FUNCTION_BLOCK SECOND_ORDER_SYSTEM_SS (* 2nd ordem system y'' + K2y' + K1y = K*Xin *)
  (* Standard: 61499-2 *)
  (* Version 11-01-12, GASR *)
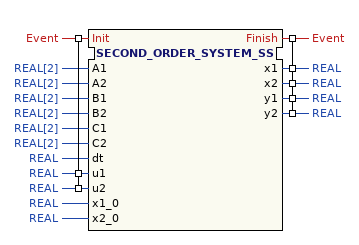
  EVENT_INPUT
    Init WITH u1, u2;
  END_EVENT
  EVENT_OUTPUT
    Finish WITH x1, x2, y1, y2;
  END_EVENT
  VAR_INPUT
    A1 : ARRAY [0..1] OF REAL; (* First row of matrix A *)
    A2 : ARRAY [0..1] OF REAL; (* Second row of matrix A *)
    B1 : ARRAY [0..1] OF REAL; (* First row of matrix B *)
    B2 : ARRAY [0..1] OF REAL; (* Second row of matrix B *)
    C1 : ARRAY [0..1] OF REAL; (* First row of matrix C *)
    C2 : ARRAY [0..1] OF REAL; (* Second row of matrix C *)
    dt : REAL;
    u1 : REAL;
    u2 : REAL;
    x1_0 : REAL; (* condicao inicial *)
    x2_0 : REAL;
  END_VAR
  VAR_OUTPUT
    x1 : REAL;
    x2 : REAL;
    y1 : REAL;
    y2 : REAL;
  END_VAR
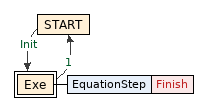
  EC_STATES
    Exe : EquationStep -> Finish;
    START;
  END_STATES
  EC_TRANSITIONS
    Exe TO START := 1;
    START TO Exe := Init;
  END_TRANSITIONS
  ALGORITHM EquationStep IN Lua: (* den[1] = b0, den[2] = b1 *)

						local function f1(X1, X2, U1, U2)
							return A1[1]*X1 + A1[2]*X2 + B1[1]*U1 + B1[2]*U2
						end

						local function f2(X1, X2, U1, U2)
							return A2[1]*X1 + A2[2]*X2 + B2[1]*U1 + B2[2]*U2
						end


						R11 = dt*f1(x1_0, x2_0, u1, u2);
						R12 = dt*f2(x1_0, x2_0, u1, u2);

						x1aux = x1_0 + 0.5*R11
						x2aux = x2_0 + 0.5*R12


						R21 = dt*f1(x1aux, x2aux, u1, u2);
						R22 = dt*f2(x1aux, x2aux, u1, u2);



						x1aux = x1aux + 0.5*R21
						x2aux = x2aux + 0.5*R22


						R31 = dt*f1(x1aux, x2aux, u1, u2);
						R32 = dt*f2(x1aux, x2aux, u1, u2);


						x1aux = x1aux + 0.5*R31
						x2aux = x2aux + 0.5*R32

						R41 = dt*f1(x1aux, x2aux, u1, u2);
						R42 = dt*f2(x1aux, x2aux, u1, u2);


						x1 = x1_0 + (1/6)*(R11 + 2*R21 + 2*R31 + R41)
						x2 = x2_0 + (1/6)*(R12 + 2*R22 + 2*R32 + R42)


						y1 = C1[1]*x1 + C1[2]*x2
						y2 = C2[1]*x1 + C2[2]*x2

						x1_0 = x1
						x2_0 = x2
  END_ALGORITHM
END_FUNCTION_BLOCK
(* other elements stored in the file *)
(* VarDeclaration Name=R11 Type=REAL *)
(* VarDeclaration Name=R12 Type=REAL *)
(* VarDeclaration Name=R21 Type=REAL *)
(* VarDeclaration Name=R22 Type=REAL *)
(* VarDeclaration Name=R31 Type=REAL *)
(* VarDeclaration Name=R32 Type=REAL *)
(* VarDeclaration Name=R41 Type=REAL *)
(* VarDeclaration Name=R42 Type=REAL *)
(* VarDeclaration Name=x1aux Type=REAL *)
(* VarDeclaration Name=x2aux Type=REAL *)
